Fanuc KAREL source: test_tof.kl

PROGRAM test_tof
%NOLOCKGROUP
%NOPAUSE = COMMAND + TPENABLE + ERROR
%UNINITVARS

%include standard.m

--uncomment to run simulation programs
--comment to stop from running

--define RUN_AVERAGING_SIM
--define RUN_SIGNAL_TEST_SIM
%define RUN_ZERO_TEST_SIM

%define AVE_MEASURE_SIM 'FR:\tof_rand.csv'
%define SIGNAL_SIM 'FR:\tof_sign.csv'
%define ZERO_SIM 'FR:\tof_zero.csv'

CONST
  SIM_TIME = 50
  NUMOFSAMPLES = 4

VAR
  last_range FROM tof1 : REAL
  is_signal FROM tof1 : BOOLEAN
  zeroed FROM tof1 : BOOLEAN
  status : INTEGER
  tof_task : BOOLEAN
  sim_task : BOOLEAN
  feed_delay : INTEGER
  range_time : INTEGER
  sim_file : STRING[16]

%include display.c.klt

-- sensor object
%class tof1('tof_sensor.klc','tof_sensor.klh','sensor_calib_test_settings.klt')

%include display.klh
%include multitask.klh
%from strings.klh %import r_to_s, b_to_s

BEGIN
  --clear display
  display__clear
  --show display
  display__show

  --set simulation program
%ifdef RUN_AVERAGING_SIM
  sim_file = AVE_MEASURE_SIM
%endif
%ifdef RUN_SIGNAL_TEST_SIM
  sim_file = SIGNAL_SIM
%endif
%ifdef RUN_ZERO_TEST_SIM
  sim_file = ZERO_SIM
%endif

  --set sample time the same as feed delay
  feed_delay = SIM_TIME

  --create tof object
  tof1__new
  --set custom sample time
  tof1__set_sample_time(feed_delay)
  --set to average ranging mode
  tof1__set_measurement_type(2)

  --total ranging task takes MAX_SAMPLES*feed_delay ms
  --to complete
  range_time = SIM_TIME*NUMOFSAMPLES

  --start ranging task
  tof_task = task__thread('tof1')

  --start simulating AI port
  sim_task = task__thread('tst_sim_tof')

%if defined(RUN_SIGNAL_TEST_SIM) || defined(RUN_AVERAGING_SIM) || defined(RUN_ZERO_TEST_SIM)
%else
%error 'Only one program flag can be on to run test.'
%endif

%ifdef RUN_SIGNAL_TEST_SIM
  DELAY 100
  -- intialize data signal
  display__print('Reading Signal : ' + b_to_s(is_signal))
%endif

  REPEAT
%ifdef RUN_AVERAGING_SIM
    display__print(r_to_s(last_range))
%endif
%ifdef RUN_SIGNAL_TEST_SIM
    IF tof1__watch_change THEN

      display__print('Reading Signal : ' + b_to_s(is_signal))
    ENDIF
%endif
%ifdef RUN_ZERO_TEST_SIM
    display__print('Reading Signal : ' + b_to_s(zeroed))
%endif
    DELAY range_time
  UNTIL(task__is_task_done('tst_sim_tof'))

  --abort ranging
  tof_task = task__abort('tof1')
  tof1__delete

  --abort sim task
  sim_task = task__abort('tst_sim_tof')

  WRITE TPDISPLAY('main task finished!',CR)

END test_tof
